// TIA Portal V17 export
// export: Created 2023-04-11T09:33:27.1487261Z, ExportSetting WithDefaults, DisplayName Totally Integrated Automation Portal, DisplayVersion V17 Update 3, DisplayName TIA Portal Openness, DisplayVersion V17 Update 3, DisplayName TIA Portal Version Control Interface, DisplayVersion V17, DisplayName SINAMICS Startdrive Advanced, DisplayVersion V17 Update2, DisplayName SINAMICS Startdrive G130, G150, S120, S150, SINAMICS MV, S210, DisplayVersion V17 Update2, DisplayName SINAMICS Startdrive G110M, G120, G120C, G120D, G120P, G115D, DisplayVersion V17 Update2, DisplayName STEP 7 Professional, DisplayVersion V17 Update 3, DisplayName STEP 7 Safety, DisplayVersion V17, DisplayName WinCC UA Professional, DisplayVersion V17 Update 3
FUNCTION_BLOCK "FB_stdCylinderJog"   // FB18, LAD
TITLE = Standart cylinder control
{ S7_Optimized_Access := 'TRUE' }
VERSION : 0.1
// stored: AutoNumber true, IsIECCheckEnabled false, IsRetainMemResEnabled false, MemoryReserve 100, SetENOAutomatically false, UDAEnableTagReadback false
   VAR_INPUT
      Double_Coil : Bool;
      Request_A : Bool;
      Request_B : Bool;
      Sensor_A : Bool;
      With_A : Bool;
      Sensor_B : Bool;
      With_B : Bool;
      Enable_A : Bool;
      Enable_B : Bool;
      Monitoring_On : Bool;
      SensorDelay_A : Time;
      SensorDelay_B : Time;
      TimeForError_A : Time;
      TimeForError_B : Time;
   END_VAR
   VAR_OUTPUT
      Out_A : Bool;
      Out_B : Bool;
      Done_A : Bool;
      Done_B : Bool;
      Error_A : Bool;
      Error_B : Bool;
      Error_moveBlock : Bool;
   END_VAR
   VAR_IN_OUT
      ABSmovement_IQ : Bool;
   END_VAR
   VAR
      FB_FaultModule_Instance { S7_SetPoint := 'True'} : "FB_faultModule";
      IEC_Timer_0_Instance { S7_SetPoint := 'True'} : TON_TIME;
      IEC_Timer_0_Instance_1 { S7_SetPoint := 'True'} : TON_TIME;
      IEC_Timer_0_Instance_2 { S7_SetPoint := 'True'} : TP_TIME;
      ABS_on : Bool;
      ABS_pulse : Bool;
      IEC_Timer_0_Instance_3 { S7_SetPoint := 'True'} : TON_TIME;
      IEC_Timer_0_Instance_4 { S7_SetPoint := 'True'} : TON_TIME;
      fillingSecondSide : Bool;
      Out_A_static : Bool;
      Out_B_static : Bool;
      IEC_Timer_0_Instance_6 { S7_SetPoint := 'True'} : TP_TIME;
      IEC_Timer_0_Instance_7 { S7_SetPoint := 'True'} : TP_TIME;
      fill_A : Bool;
      fill_B : Bool;
      IEC_Timer_0_Instance_9 { S7_SetPoint := 'True'} : TON_TIME;
      IEC_Timer_0_Instance_8 { S7_SetPoint := 'True'} : TON_TIME;
   END_VAR
BEGIN

REGION Network 1: ABS pulse generate
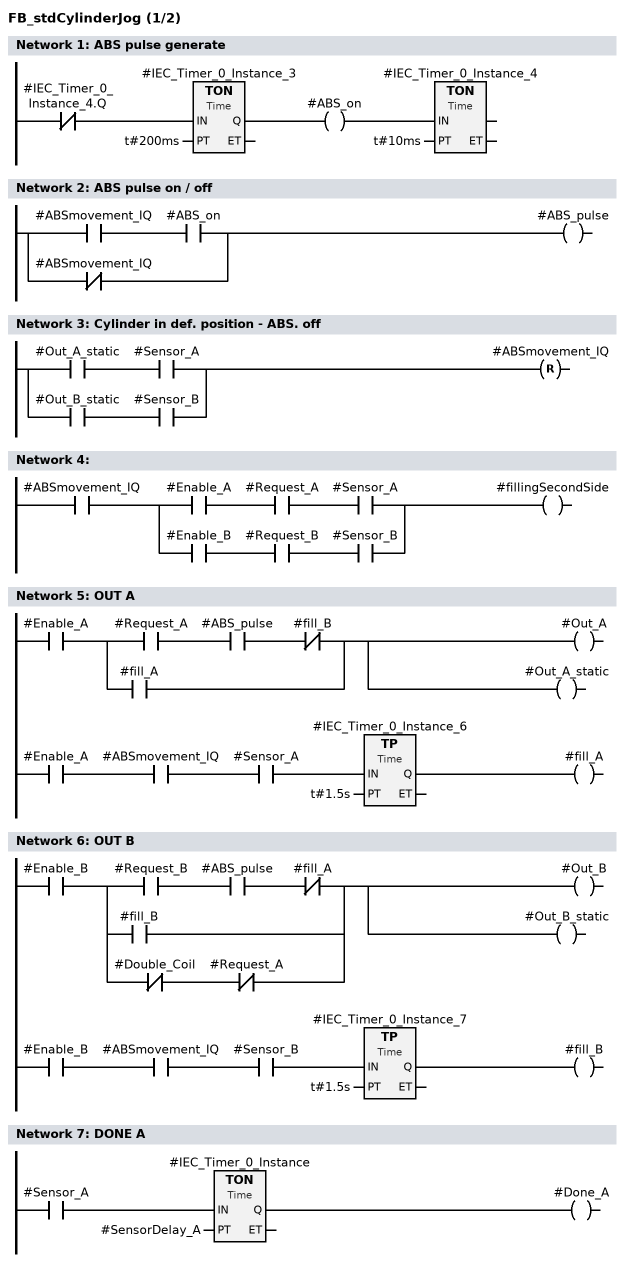
   RUNG wire#powerrail
      I_Contact( #IEC_Timer_0_Instance_4.Q )
      { S7_Templates := "time_type := Time" } #IEC_Timer_0_Instance_3.TON(pt := t#200ms, et =>)
      Coil( #ABS_on )
      { S7_Templates := "time_type := Time" } #IEC_Timer_0_Instance_4.TON(pt := t#10ms, et =>)
   END_RUNG
   // the same network as SCL:
   #IEC_Timer_0_Instance_3(IN := NOT #IEC_Timer_0_Instance_4.Q, PT := t#200ms);   // TON
   #ABS_on := #IEC_Timer_0_Instance_3.Q;
   #IEC_Timer_0_Instance_4(IN := #IEC_Timer_0_Instance_3.Q, PT := t#10ms);   // TON
END_REGION

REGION Network 2: ABS pulse on / off
   RUNG wire#powerrail
      Contact( #ABSmovement_IQ )
      Contact( #ABS_on )
      wire#w1
      Coil( #ABS_pulse )
   END_RUNG
   RUNG wire#powerrail
      I_Contact( #ABSmovement_IQ )
   END_RUNG wire#w1
   // the same network as SCL:
   #ABS_pulse := (#ABSmovement_IQ AND #ABS_on) OR NOT #ABSmovement_IQ;
END_REGION

REGION Network 3: Cylinder in def. position - ABS. off
   RUNG wire#powerrail
      Contact( #Out_A_static )
      Contact( #Sensor_A )
      wire#w1
      R_Coil( #ABSmovement_IQ )
   END_RUNG
   RUNG wire#powerrail
      Contact( #Out_B_static )
      Contact( #Sensor_B )
   END_RUNG wire#w1
   // the same network as SCL:
   IF (#Out_A_static AND #Sensor_A) OR (#Out_B_static AND #Sensor_B) THEN #ABSmovement_IQ := FALSE; END_IF;
END_REGION

REGION Network 4
   RUNG wire#powerrail
      Contact( #ABSmovement_IQ )
      wire#w1
      Contact( #Enable_A )
      Contact( #Request_A )
      Contact( #Sensor_A )
      wire#w2
      Coil( #fillingSecondSide )
   END_RUNG
   RUNG wire#w1
      Contact( #Enable_B )
      Contact( #Request_B )
      Contact( #Sensor_B )
   END_RUNG wire#w2
   // the same network as SCL:
   #fillingSecondSide := #ABSmovement_IQ AND ((#Enable_A AND #Request_A AND #Sensor_A) OR (#Enable_B AND #Request_B AND #Sensor_B));
END_REGION

REGION Network 5: OUT A
   RUNG wire#powerrail
      Contact( #Enable_A )
      wire#w1
      Contact( #Request_A )
      Contact( #ABS_pulse )
      I_Contact( #fill_B )
      wire#w2
      Coil( #Out_A )
   END_RUNG
   RUNG wire#w1
      Contact( #fill_A )
   END_RUNG wire#w2
   RUNG wire#w2
      Coil( #Out_A_static )
   END_RUNG
   RUNG wire#powerrail
      Contact( #Enable_A )
      Contact( #ABSmovement_IQ )
      Contact( #Sensor_A )
      { S7_Templates := "time_type := Time" } #IEC_Timer_0_Instance_6.TP(pt := t#1.5s, et =>)
      Coil( #fill_A )
   END_RUNG
   // the same network as SCL:
   #Out_A := #Enable_A AND ((#Request_A AND #ABS_pulse AND NOT #fill_B) OR #fill_A);
   #Out_A_static := #Out_A;
   #IEC_Timer_0_Instance_6(IN := #Enable_A AND #ABSmovement_IQ AND #Sensor_A, PT := t#1.5s);   // TP
   #fill_A := #IEC_Timer_0_Instance_6.Q;
END_REGION

REGION Network 6: OUT B
   RUNG wire#powerrail
      Contact( #Enable_B )
      wire#w1
      Contact( #Request_B )
      Contact( #ABS_pulse )
      I_Contact( #fill_A )
      wire#w2
      Coil( #Out_B )
   END_RUNG
   RUNG wire#w1
      Contact( #fill_B )
   END_RUNG wire#w2
   RUNG wire#w1
      I_Contact( #Double_Coil )
      I_Contact( #Request_A )
   END_RUNG wire#w2
   RUNG wire#w2
      Coil( #Out_B_static )
   END_RUNG
   RUNG wire#powerrail
      Contact( #Enable_B )
      Contact( #ABSmovement_IQ )
      Contact( #Sensor_B )
      { S7_Templates := "time_type := Time" } #IEC_Timer_0_Instance_7.TP(pt := t#1.5s, et =>)
      Coil( #fill_B )
   END_RUNG
   // the same network as SCL:
   #Out_B := #Enable_B AND ((#Request_B AND #ABS_pulse AND NOT #fill_A) OR #fill_B OR (NOT #Double_Coil AND NOT #Request_A));
   #Out_B_static := #Out_B;
   #IEC_Timer_0_Instance_7(IN := #Enable_B AND #ABSmovement_IQ AND #Sensor_B, PT := t#1.5s);   // TP
   #fill_B := #IEC_Timer_0_Instance_7.Q;
END_REGION

REGION Network 7: DONE A
   RUNG wire#powerrail
      Contact( #Sensor_A )
      { S7_Templates := "time_type := Time" } #IEC_Timer_0_Instance.TON(pt := #SensorDelay_A, et =>)
      Coil( #Done_A )
   END_RUNG
   // the same network as SCL:
   #IEC_Timer_0_Instance(IN := #Sensor_A, PT := #SensorDelay_A);   // TON
   #Done_A := #IEC_Timer_0_Instance.Q;
END_REGION

REGION Network 8: DONE B
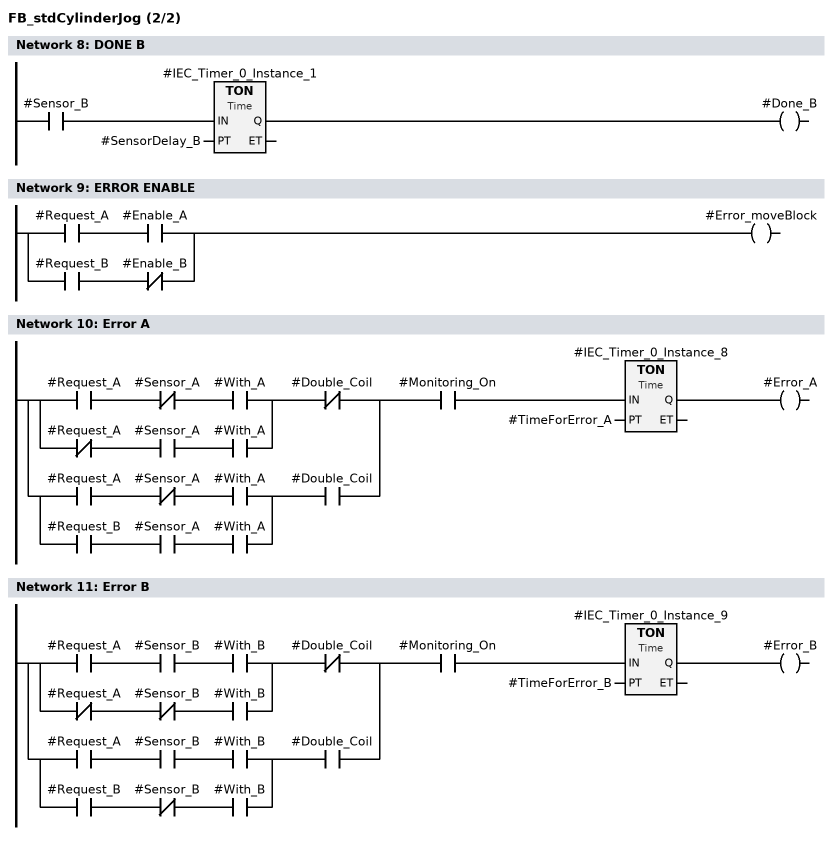
   RUNG wire#powerrail
      Contact( #Sensor_B )
      { S7_Templates := "time_type := Time" } #IEC_Timer_0_Instance_1.TON(pt := #SensorDelay_B, et =>)
      Coil( #Done_B )
   END_RUNG
   // the same network as SCL:
   #IEC_Timer_0_Instance_1(IN := #Sensor_B, PT := #SensorDelay_B);   // TON
   #Done_B := #IEC_Timer_0_Instance_1.Q;
END_REGION

REGION Network 9: ERROR ENABLE
   RUNG wire#powerrail
      Contact( #Request_A )
      Contact( #Enable_A )
      wire#w1
      Coil( #Error_moveBlock )
   END_RUNG
   RUNG wire#powerrail
      Contact( #Request_B )
      I_Contact( #Enable_B )
   END_RUNG wire#w1
   // the same network as SCL:
   #Error_moveBlock := (#Request_A AND #Enable_A) OR (#Request_B AND NOT #Enable_B);
END_REGION

REGION Network 10: Error A
   RUNG wire#powerrail
      Contact( #Request_A )
      I_Contact( #Sensor_A )
      Contact( #With_A )
      wire#w1
      I_Contact( #Double_Coil )
      wire#w2
      Contact( #Monitoring_On )
      { S7_Templates := "time_type := Time" } #IEC_Timer_0_Instance_8.TON(pt := #TimeForError_A, et =>)
      Coil( #Error_A )
   END_RUNG
   RUNG wire#powerrail
      I_Contact( #Request_A )
      Contact( #Sensor_A )
      Contact( #With_A )
   END_RUNG wire#w1
   RUNG wire#powerrail
      Contact( #Request_A )
      I_Contact( #Sensor_A )
      Contact( #With_A )
      wire#w3
      Contact( #Double_Coil )
   END_RUNG wire#w2
   RUNG wire#powerrail
      Contact( #Request_B )
      Contact( #Sensor_A )
      Contact( #With_A )
   END_RUNG wire#w3
   // the same network as SCL:
   #IEC_Timer_0_Instance_8(IN := ((((#Request_A AND NOT #Sensor_A AND #With_A) OR (NOT #Request_A AND #Sensor_A AND #With_A)) AND NOT #Double_Coil) OR (((#Request_A AND NOT #Sensor_A AND #With_A) OR (#Request_B AND #Sensor_A AND #With_A)) AND #Double_Coil)) AND #Monitoring_On,   // TON
                           PT := #TimeForError_A);
   #Error_A := #IEC_Timer_0_Instance_8.Q;
END_REGION

REGION Network 11: Error B
   RUNG wire#powerrail
      Contact( #Request_A )
      Contact( #Sensor_B )
      Contact( #With_B )
      wire#w1
      I_Contact( #Double_Coil )
      wire#w2
      Contact( #Monitoring_On )
      { S7_Templates := "time_type := Time" } #IEC_Timer_0_Instance_9.TON(pt := #TimeForError_B, et =>)
      Coil( #Error_B )
   END_RUNG
   RUNG wire#powerrail
      I_Contact( #Request_A )
      I_Contact( #Sensor_B )
      Contact( #With_B )
   END_RUNG wire#w1
   RUNG wire#powerrail
      Contact( #Request_A )
      Contact( #Sensor_B )
      Contact( #With_B )
      wire#w3
      Contact( #Double_Coil )
   END_RUNG wire#w2
   RUNG wire#powerrail
      Contact( #Request_B )
      I_Contact( #Sensor_B )
      Contact( #With_B )
   END_RUNG wire#w3
   // the same network as SCL:
   #IEC_Timer_0_Instance_9(IN := ((((#Request_A AND #Sensor_B AND #With_B) OR (NOT #Request_A AND NOT #Sensor_B AND #With_B)) AND NOT #Double_Coil) OR (((#Request_A AND #Sensor_B AND #With_B) OR (#Request_B AND NOT #Sensor_B AND #With_B)) AND #Double_Coil)) AND #Monitoring_On,   // TON
                           PT := #TimeForError_B);
   #Error_B := #IEC_Timer_0_Instance_9.Q;
END_REGION
END_FUNCTION_BLOCK
